Fanuc KAREL source: kt00036.KL

-- PROVISIONAL review KL for V770-1; original PC SHA256 b76e61edf7f14c95fffe789d8e4807d699a58e1c85727349095578e7829d8b87
-- Incomplete behavior may be omitted. Consult companion uncertainty JSON. Do not deploy.
PROGRAM KT00036
%NOLOCKGROUP
VAR
  I1 : INTEGER
  R2 : REAL
  OUT : REAL
BEGIN
  -- UNRESOLVED_PC offsets 5-16; opcodes 2E,23
  -- UNRESOLVED_PC offsets 21-32; opcodes 2E,23
  -- UNRESOLVED_PC offsets 37-59; opcodes 21,21,29,64,29,6A,23
  -- UNRESOLVED_PC offsets 64-68; opcodes 7F
END KT00036
